(* PLC project LD_TEST, Beremiz BREMIZ 1 *)
(* stored: contentDescription This tests SFC language, companyURL www.beremiz.org, productRelease 1, creationDateTime 2007-07-07 11:58:26 *)

PROGRAM MAIN_TEST
  VAR
    QX1 AT %QX1 : BOOL := FALSE;
    QX2 AT %QX2 : BOOL := TRUE;
    QX3 AT %QX3 : BOOL;
    IX1 AT %IX1 : BOOL;
    IX2 AT %IX2 : BOOL;
    IX3 AT %IX3 : BOOL;
  END_VAR

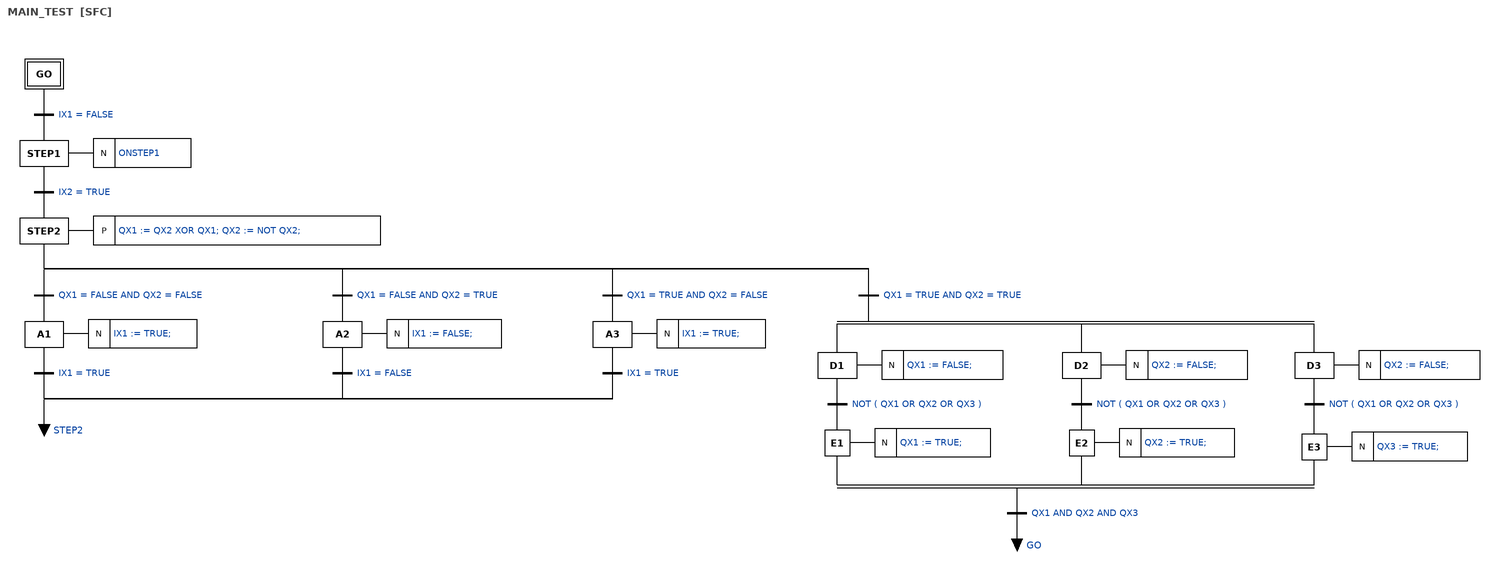
INITIAL_STEP GO:
END_STEP
TRANSITION FROM GO TO STEP1
  := IX1 = FALSE;
END_TRANSITION
STEP STEP1:
  ONSTEP1(N);
END_STEP
TRANSITION FROM STEP1 TO STEP2
  := IX2 = TRUE;
END_TRANSITION
STEP STEP2:
  STEP2_INLINE1(P);
END_STEP
ACTION STEP2_INLINE1:
  QX1 := QX2 XOR QX1; QX2 := NOT QX2;
END_ACTION
TRANSITION FROM STEP2 TO A1
  := QX1 = FALSE AND QX2 = FALSE;
END_TRANSITION
TRANSITION FROM STEP2 TO (D1, D2, D3)
  := QX1 = TRUE AND QX2 = TRUE;
END_TRANSITION
TRANSITION FROM STEP2 TO A3
  := QX1 = TRUE AND QX2 = FALSE;
END_TRANSITION
TRANSITION FROM STEP2 TO A2
  := QX1 = FALSE AND QX2 = TRUE;
END_TRANSITION
STEP A1:
  A1_INLINE2(N);
END_STEP
ACTION A1_INLINE2:
  IX1 := TRUE;
END_ACTION
TRANSITION FROM A1 TO STEP2
  := IX1 = TRUE;
END_TRANSITION
STEP A2:
  A2_INLINE3(N);
END_STEP
ACTION A2_INLINE3:
  IX1 := FALSE;
END_ACTION
TRANSITION FROM A2 TO STEP2
  := IX1 = FALSE;
END_TRANSITION
STEP A3:
  A3_INLINE4(N);
END_STEP
ACTION A3_INLINE4:
  IX1 := TRUE;
END_ACTION
TRANSITION FROM A3 TO STEP2
  := IX1 = TRUE;
END_TRANSITION
STEP D1:
  D1_INLINE5(N);
END_STEP
ACTION D1_INLINE5:
  QX1 := FALSE;
END_ACTION
TRANSITION FROM D1 TO E1
  := NOT ( QX1 OR QX2 OR QX3 );
END_TRANSITION
STEP D2:
  D2_INLINE6(N);
END_STEP
ACTION D2_INLINE6:
  QX2 := FALSE;
END_ACTION
TRANSITION FROM D2 TO E2
  := NOT ( QX1 OR QX2 OR QX3 );
END_TRANSITION
STEP D3:
  D3_INLINE7(N);
END_STEP
ACTION D3_INLINE7:
  QX2 := FALSE;
END_ACTION
TRANSITION FROM D3 TO E3
  := NOT ( QX1 OR QX2 OR QX3 );
END_TRANSITION
STEP E1:
  E1_INLINE8(N);
END_STEP
ACTION E1_INLINE8:
  QX1 := TRUE;
END_ACTION
TRANSITION FROM (E1, E2, E3) TO GO
  := QX1 AND QX2 AND QX3;
END_TRANSITION
STEP E2:
  E2_INLINE9(N);
END_STEP
ACTION E2_INLINE9:
  QX2 := TRUE;
END_ACTION
STEP E3:
  E3_INLINE10(N);
END_STEP
ACTION E3_INLINE10:
  QX3 := TRUE;
END_ACTION

ACTION ONSTEP1:
QX1 := TRUE;
QX2 := TRUE;
              
END_ACTION
END_PROGRAM

CONFIGURATION STD_CONF
  RESOURCE STD_RESSOURCE ON PLC
    TASK STD_TASK(INTERVAL := 00:00:00.100000, PRIORITY := 0);
    PROGRAM MAIN_INSTANCE : MAIN_TEST;
  END_RESOURCE
END_CONFIGURATION
